TYPE E_DilPrepareMode :
(
	ForAspirate := 0,
	ForDispense := 1
)USINT;
END_TYPE

(* stored: Version 1.1.0.1, ProductVersion 3.1.4020.12
   DUT E_DilPrepareMode: Id {37528f9d-faf5-4857-b422-f66bf905a1e2} *)
